% RSLogix 500 project timer.RSS, saved by version 8.30.00.16 %
PROJECT "UNTITLED"    % processor: MicroLogix 1000 %

PROGRAM FILES
  LAD 2 "MAIN_PROG"  9 rungs
  LAD 3 "USER_FAULT"  1 rungs
  LAD 4 "HSC_INT"  1 rungs
  LAD 5 "STI_INT"  1 rungs
  LAD 6, 7, 8, 9, 10, 11, 12, 13, 14, 15, 16: only END

DATA FILES
  O0 OUTPUT  1 elements
  I1 INPUT  2 elements
  S2 STATUS  33 elements
  B3 BINARY  32 elements
  T4 TIMER  40 elements
  C5 COUNTER  32 elements
  R6 CONTROL  16 elements
  N7 INTEGER  105 elements

LADDER 2 "MAIN_PROG"
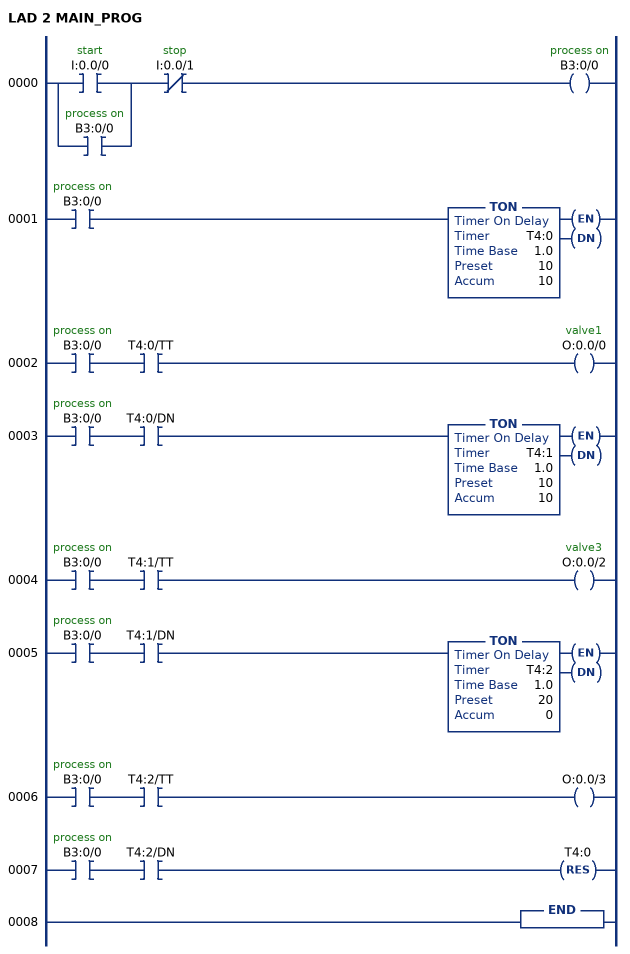
% Rung: 0 %
SOR BST XIC I:0.0/0 NXB XIC B3:0/0 BND XIO I:0.0/1 OTE B3:0/0 EOR
%   I:0.0/0  "start" %
%   B3:0/0  "process on" %
%   I:0.0/1  "stop" %
% Rung: 1 %
SOR XIC B3:0/0 TON T4:0 1.0 10 10 EOR
%   B3:0/0  "process on" %
% Rung: 2 %
SOR XIC B3:0/0 XIC T4:0/TT OTE O:0.0/0 EOR
%   B3:0/0  "process on" %
%   O:0.0/0  "valve1" %
% Rung: 3 %
SOR XIC B3:0/0 XIC T4:0/DN TON T4:1 1.0 10 10 EOR
%   B3:0/0  "process on" %
% Rung: 4 %
SOR XIC B3:0/0 XIC T4:1/TT OTE O:0.0/2 EOR
%   B3:0/0  "process on" %
%   O:0.0/2  "valve3" %
% Rung: 5 %
SOR XIC B3:0/0 XIC T4:1/DN TON T4:2 1.0 20 0 EOR
%   B3:0/0  "process on" %
% Rung: 6 %
SOR XIC B3:0/0 XIC T4:2/TT OTE O:0.0/3 EOR
%   B3:0/0  "process on" %
% Rung: 7 %
SOR XIC B3:0/0 XIC T4:2/DN RES T4:0 EOR
%   B3:0/0  "process on" %
% Rung: 8 %
SOR END EOR

OTHER DOCUMENTED ADDRESSES
  O:0.0/1  "valve2"

DATA TABLE (non-zero values as saved)
DATA B3
% B3:0 % 0X0001 0X0000 0X0000 0X0000 0X0000 0X0000 0X0000 0X0000 0X0000 0X0000
DATA T4
% .PRE .ACC %
% T4:0 % 10 10
% T4:1 % 10 10
% T4:2 % 20 0
